FUNCTION rot2AngAxis : bool
VAR_IN_OUT CONSTANT
	rot : Mat3d;
END_VAR
VAR_OUTPUT
	angle: LREAL;
	axis : Vec3d;
END_VAR
VAR
	tmp:LREAL;
END_VAR

tmp:=LIMIT(-1, (rot[1,1]+rot[2,2]+rot[3,3]-1)/2 , 1);
angle := ACOS(tmp);

// no rotation
IF ABS(angle)<g_smallAng THEN
	angle :=0;
	axis[1]:=1;
	axis[2]:=0;
	axis[3]:=0;
// rotate pi
ELSIF ABS(angle-pi)< g_smallAng THEN
	angle :=PI;
	axis[1]:=SQRT((rot[1,1]+1)/2);
	axis[2]:=SQRT((rot[2,2]+1)/2);
	axis[3]:=SQRT((rot[3,3]+1)/2);
	IF axis[1]>g_smallNum THEN
		axis[2]:=0.5*rot[1,2]/axis[1];
		axis[3]:=0.5*rot[1,3]/axis[1];
	ELSIF axis[2]>g_smallNum THEN
		axis[1]:=0.5*rot[2,1]/axis[2];
		axis[3]:=0.5*rot[2,3]/axis[2];
	ELSE
		axis[1]:=0.5*rot[3,1]/axis[3];
		axis[2]:=0.5*rot[3,2]/axis[3];
	END_IF
// others
ELSE
	tmp:=2*SIN(angle);
	axis[1]:=(rot[3,2]-rot[2,3])/tmp;
	axis[2]:=(rot[1,3]-rot[3,1])/tmp;
	axis[3]:=(rot[2,1]-rot[1,2])/tmp;
END_IF

// normalize
normalize(axis);

END_FUNCTION

(* stored: Version 1.1.0.1, ProductVersion 3.1.4024.11
   POU rot2AngAxis: Id {2ad75c44-ef95-44e4-9940-6f53f74e7147}, SpecialFunc None *)
